TYPE WaferInspection :
STRUCT
	SKU : SKURecipe;
	Cavities : CavityRecipe;
	Wafer : WaferRecipe;
	Camera : CameraRecipe;
END_STRUCT
END_TYPE

(* stored: Version 1.1.0.1
   DUT WaferInspection: Id {22b68b08-2649-43f3-9892-88bd54dffb13} *)
